FUNCTION FUNC_Add : INT
VAR_INPUT
  nA : INT;
  nB : INT;
END_VAR

FUNC_Add := nA + nB;

END_FUNCTION

(* stored: Version 1.1.0.1, ProductVersion 3.1.4024.12
   POU FUNC_Add: Id {b1c2d3e4-f5a6-7890-abcd-ef1234567891}, SpecialFunc None *)
